TYPE ST_MC_Status :
STRUCT
	
	Status		:	BOOL;
	Done		:	BOOL;
	Busy		:	BOOL;
	Error		:	BOOL;
	Active		:	BOOL;
	CmdAborted	:	BOOL;
	InVelocity	:	BOOL;
	ErrrorID	:	UDINT;

END_STRUCT
END_TYPE

(* stored: Version 1.1.0.1, ProductVersion 3.1.4024.11
   DUT ST_MC_Status: Id {450459eb-5d3c-4b77-9e66-da445ad8a02b} *)
